PROGRAM MAIN
VAR
END_VAR

END_PROGRAM

(* stored: Version 1.1.0.1
   POU MAIN: Id {2887826a-8a5a-40e3-a0d6-624a25de52e5} *)
